{attribute 'GeneratedUsingTerminal: EK1100-0000-0018'}
{attribute addProperty BoxType "EK1100-0000-0018"}
{attribute addProperty Id "Beckhoff_ELM35xxEK1122Beckhoff_ELM35xxEK1122_0F7152EB2A_0001_ELM3502_0000_0016ELM3502_3D4ED79F42A_0002_ELM3502_0000_0017ELM3502_3D4ED79F42A_0003_ELM3502_0000_0018ELM3502_3D4ED79F42A_0004_ELM3502_0000_0019ELM3502_3D4ED79F42A_0005_ELM3504_0000_0016ELM3504_177D76D464A_0006_ELM3504_0000_0017ELM3504_177D76D464A_0007_ELM3504_0000_0018ELM3504_177D76D464A_0008_ELM3504_0000_0019ELM3504_177D76D464"}
{attribute addProperty CRC "4070861946"}
{attribute addProperty Size "426"}
TYPE Beckhoff_ELM35xx_F2A46C7A EXTENDS EK1100_1FC0878B :
STRUCT
	{attribute addProperty Name "Beckhoff_ELM35xxEK1122"}
	{attribute addProperty PreviousPort "Beckhoff ELM35xx : B"}
	Beckhoff_ELM35xxEK1122 : Beckhoff_ELM35xxEK1122_0F7152EB;
	{attribute addProperty Name "A_0001_ELM3502_0000_0016"}
	{attribute addProperty PreviousPort "Beckhoff ELM35xxEK1122 : C"}
	A_0001_ELM3502_0000_0016 : ELM3502_3D4ED79F;
	{attribute addProperty Name "A_0002_ELM3502_0000_0017"}
	{attribute addProperty PreviousPort "A_0001(ELM3502-0000-0016) : B"}
	A_0002_ELM3502_0000_0017 : ELM3502_3D4ED79F;
	{attribute addProperty Name "A_0003_ELM3502_0000_0018"}
	{attribute addProperty PreviousPort "A_0002(ELM3502-0000-0017) : B"}
	A_0003_ELM3502_0000_0018 : ELM3502_3D4ED79F;
	{attribute addProperty Name "A_0004_ELM3502_0000_0019"}
	{attribute addProperty PreviousPort "A_0003(ELM3502-0000-0018) : B"}
	A_0004_ELM3502_0000_0019 : ELM3502_3D4ED79F;
	{attribute addProperty Name "A_0005_ELM3504_0000_0016"}
	{attribute addProperty PreviousPort "A_0004(ELM3502-0000-0019) : B"}
	A_0005_ELM3504_0000_0016 : ELM3504_177D76D4;
	{attribute addProperty Name "A_0006_ELM3504_0000_0017"}
	{attribute addProperty PreviousPort "A_0005(ELM3504-0000-0016) : B"}
	A_0006_ELM3504_0000_0017 : ELM3504_177D76D4;
	{attribute addProperty Name "A_0007_ELM3504_0000_0018"}
	{attribute addProperty PreviousPort "A_0006(ELM3504-0000-0017) : B"}
	A_0007_ELM3504_0000_0018 : ELM3504_177D76D4;
	{attribute addProperty Name "A_0008_ELM3504_0000_0019"}
	{attribute addProperty PreviousPort "A_0007(ELM3504-0000-0018) : B"}
	A_0008_ELM3504_0000_0019 : ELM3504_177D76D4;
END_STRUCT
END_TYPE

(* stored: Version 1.2.0.0, ProductVersion 3.1.4024.9
   DUT Beckhoff_ELM35xx_F2A46C7A: Id {a49d70b6-87c1-462e-a004-eeac8da4ab5b} *)
